FUNCTION_BLOCK EV_Piston (* Typed view of Piston's state channel (inputs and holder) *)
  (* Standard: 61499-2 *)
  (* Version 0.1, 2026-09-28, Project contributors, AAU Smart Production Lab *)
  PACKAGE stoppering;
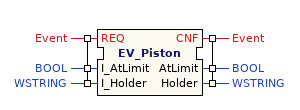
  EVENT_INPUT
    REQ WITH I_AtLimit, I_Holder;
  END_EVENT
  EVENT_OUTPUT
    CNF WITH AtLimit, Holder;
  END_EVENT
  VAR_INPUT
    I_AtLimit : BOOL;
    I_Holder : WSTRING;
  END_VAR
  VAR_OUTPUT
    AtLimit : BOOL;
    Holder : WSTRING;
  END_VAR
  EC_STATES
    REQ : REQ -> CNF;
  END_STATES
  ALGORITHM REQ IN ST:
AtLimit := I_AtLimit;
Holder := I_Holder;
  END_ALGORITHM
END_FUNCTION_BLOCK
